FUNCTION_BLOCK NoCmd (* CAT Function Block Type *)
  (* Standard: 61499-2 *)
  (* Version 0.0, 6/7/2026, Schneider Electric, template *)
  PACKAGE SE.Nereda;
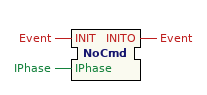
  EVENT_INPUT
    INIT;
  END_EVENT
  EVENT_OUTPUT
    INITO;
  END_EVENT
  SOCKETS
    IPhase : IPhase;
  END_SOCKETS
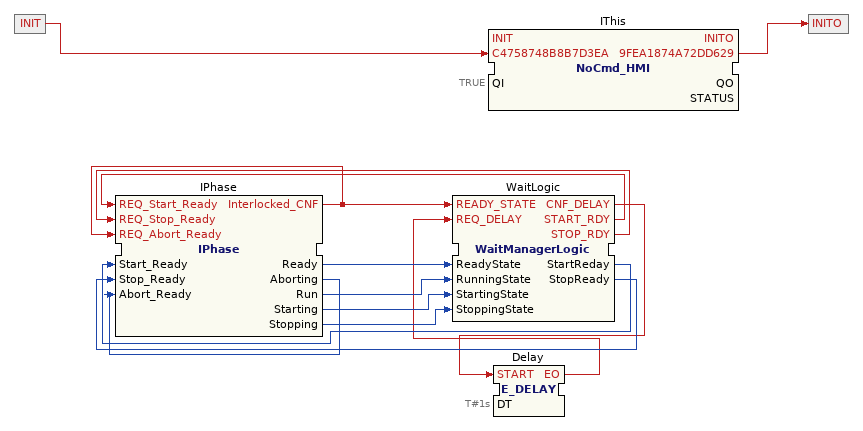
  (* 01 - FUNCTIONNAL INPUT INTERFACE *)
  (* 00 - INITIALIZATION *)
  (* 05 - LOGIC *)
  (* 06 - HMI INTERFACE *)
  (* 03 - FIELD INTERFACE *)
  (* 02 - FUNCTIONNAL OUTPUT INTERFACE *)
  FBS
    IThis : NoCmd_HMI(QI := TRUE);
    WaitLogic : WaitManagerLogic;
    Delay : E_DELAY(DT := T#1s);
  END_FBS
  EVENT_CONNECTIONS
    INIT TO IThis.C4758748B8B7D3EA;
    IThis.9FEA1874A72DD629 TO INITO;
    IPhase.Interlocked_CNF TO WaitLogic.READY_STATE;
    WaitLogic.CNF_DELAY TO Delay.START;
    Delay.EO TO WaitLogic.REQ_DELAY;
    WaitLogic.START_RDY TO IPhase.REQ_Start_Ready;
    WaitLogic.STOP_RDY TO IPhase.REQ_Stop_Ready;
    IPhase.Interlocked_CNF TO IPhase.REQ_Abort_Ready;
  END_CONNECTIONS
  DATA_CONNECTIONS
    IPhase.Ready TO WaitLogic.ReadyState;
    WaitLogic.StartReday TO IPhase.Start_Ready;
    WaitLogic.StopReady TO IPhase.Stop_Ready;
    IPhase.Aborting TO IPhase.Abort_Ready;
    IPhase.Run TO WaitLogic.RunningState;
    IPhase.Starting TO WaitLogic.StartingState;
    IPhase.Stopping TO WaitLogic.StoppingState;
  END_CONNECTIONS
END_FUNCTION_BLOCK
